                       //increase tree index to access next element 
                       #statIndexTreeArray += SINT_TO_UINT(#INCREMENT_BY_ONE);

                       //element was closed, pop index from stack
                       #statStackIndex -= SINT_TO_INT(#DECREMENT_BY_ONE);

                       //Set state, that should be executed after writing
                       #statFbNextState := #FB_STATE_CLOSE_STACK_ELEMENT;

                     ELSE
                       //close element with syntax key > as next element is child
                       // statInfoToWrite --> >
                       #statInfoToWrite := #XML_KEY_CLOSE_GREATER;
                       //Set state, that should be executed after writing
                       #statFbNextState := #FB_STATE_NEXT_ELEMENT;
                       //increase tree index to access next element 
                       #statIndexTreeArray += SINT_TO_UINT(#INCREMENT_BY_ONE);
                     END_IF;
                   END_IF;
                   //END Element
                 END_REGION ELEMENT

               ELSE // Undefined type provided
                 REGION UNDEFINED TYPE
                   #statStatus := #ERR_UNDEFINED_TYPE;
                 END_REGION UNDEFINED TYPE
             END_CASE;

             //Move to state Write
             #statFbState := #FB_STATE_WRITE_TO_XML;

           END_REGION WRITE VALUE

         #FB_STATE_CLOSE_STACK_ELEMENT: //Close Open Stack Elements
           REGION CLOSE ELEMENT FROM STACK
             //close element with syntax </key>

             IF #statStackIndex >= 0 THEN //more open elements available, not all elements are closed

               //statInfoToWrite --> </key>
               #statInfoToWrite := CONCAT(IN1 := #XML_KEY_OPEN,
                                          IN2 := #XML_KEY_CLOSE_SLASH,
                                          IN3 := #tree[#statStackIndexOpenElement[#statStackIndex]].key,
                                          IN4 := #XML_KEY_CLOSE_GREATER);

               //pop element from stack 
               #statStackIndex -= SINT_TO_INT(#DECREMENT_BY_ONE);

               IF #statStackIndex >= 0 THEN //more open elements available, not all elements are closed
                 //look at current stack item depth, if next tree element has 
                 IF NOT #statIsLastElement AND #tree[#statStackIndexOpenElement[#statStackIndex]].depth < #tree[#statIndexTreeArray + #NEXT_INDEX].depth THEN
                   //move to next element
                   #statFbNextState := #FB_STATE_NEXT_ELEMENT;
                   //increase tree index to access next element 
                   #statIndexTreeArray += SINT_TO_UINT(#INCREMENT_BY_ONE);
                 ELSE
                   //do nothing and return to fb state close element 
                   #statFbNextState := #FB_STATE_CLOSE_STACK_ELEMENT;
                 END_IF;

               ELSE
                 //no more open Elements, last Element was closed
                 #statIsLastElement := TRUE;

                 //only if this flag is set, can writer be finished
                 #statLastElementIsClosed := TRUE;

               END_IF;

             ELSE
               //no more open Elements, last Element was closed
               #statIsLastElement := TRUE;

               //only if this flag is set, can writer be finished
               #statLastElementIsClosed := TRUE;

             END_IF;
             //Move to state Write
             #statFbState := #FB_STATE_WRITE_TO_XML;
           END_REGION CLOSE ELEMENT FROM STACK

         #FB_STATE_WRITE_TO_XML: // Write to Byte Array
           REGION WRITE TO XML                
             //add information to xml byte array
             IF ((INT_TO_UINT(LEN(#statInfoToWrite)) + #statIndexXmlByteArray) < #statXmlByteLen) THEN
               Strg_TO_Chars(Strg := #statInfoToWrite,
                             pChars := #statIndexXmlByteArray,
                             Cnt => #tempCntCharsAdded,
                             Chars := #xmlByteArray);

               //move index of byte array 
               #statIndexXmlByteArray += #tempCntCharsAdded;
               //move to next state previously allocated
               #statFbState := #statFbNextState;
             ELSE // Error: Index out of bounds
               #statStatus := #ERR_XML_OUT_OF_BOUNDS;
             END_IF;

             IF #statLastElementIsClosed THEN
               //writer has written last information and execution is done
               #statStatus := #STATUS_EXECUTION_FINISHED;
               //current index equals count/size of xml byte array
               #statCount := #statIndexXmlByteArray;
             END_IF;
           END_REGION WRITE TO XML

         ELSE // Undefined state in state machine reached
           REGION UNDEFINED STATE
             #statStatus := #ERR_UNDEFINED_STATE;
           END_REGION UNDEFINED STATE                

       END_CASE;
       //Leave state machine if one of the following condition is true
       //1. state has not changed
       //2. error has occured
       //3. watchdog timer expired 
       //4. execution has finished
       // otherwise stay in state machine
     UNTIL (#statFbPreviousState = #statFbState OR #statStatus.%X15
       OR #instWatchdog.Q OR #statStatus = #STATUS_EXECUTION_FINISHED)
     END_REPEAT;
   END_REGION STATE_MACHINE

   REGION OUTPUTS
     // Write outputs
     IF (#statStatus = #STATUS_EXECUTION_FINISHED) AND (#statDone = FALSE) THEN // Execution finished without errors
       REGION EXECUTION FINSIHED
         #statDone := TRUE;
         #statBusy := FALSE;
         #statError := FALSE;
         // execution aborted --> set state no processing
         #statFbState := #FB_STATE_NO_PROCESSING;
       END_REGION EXECUTION FINSIHED

     ELSIF (#statStatus.%X15 = TRUE) AND (#statError = FALSE) THEN // Error occurred (#statStatus is 16#8000 to 16#FFFF)
       REGION ERROR OCCURED
         #statDone := FALSE;
         #statBusy := FALSE;
         #statError := TRUE;
         // execution aborted --> set state no processing
         #statFbState := #FB_STATE_NO_PROCESSING;
       END_REGION ERROR OCCURED

     ELSIF (#tempExecute = FALSE) AND ((#statDone = TRUE) OR (#statError = TRUE)) THEN // Reset outputs
       REGION EXECUTE RESETTED
         #statDone := FALSE;
         #statBusy := FALSE;
         #statError := FALSE;
         #statStatus := #STATUS_NO_CALL;
         // Reset application specific outputs
         #statCount := 0;
       END_REGION EXECUTE RESETTED
     END_IF;

     REGION WRITE STATIC VALUES TO OUTPUTS
       #done := #statDone;
       #busy := #statBusy;
       #error := #statError;
       #status := #statStatus;
       //  ENO mechanism is not used 
       ENO := TRUE;
       // Write application specific static values to outputs
       #count := #statCount;
     END_REGION WRITE STATIC VALUES TO OUTPUTS
   END_REGION OUTPUTS
END_FUNCTION_BLOCK

// folder: LStream/Utilities

FUNCTION "LStream_FindStringInByteCharArrayAdv" : DInt   // FC2, SCL
TITLE = LStream_FindStringInCharArrayAdv
{ S7_Optimized_Access := 'TRUE' }
AUTHOR : DI_FA_S_SUP_EuC
FAMILY : LStream
VERSION : 1.0
// Finds string in char array
   VAR_INPUT
      searchFor : String;   // Text that is searched for
      startPosition : DInt;   // Start position in array
   END_VAR
   VAR_IN_OUT
      searchIn : Array[*] of Byte;   // Array of Char to search in
   END_VAR
   VAR_TEMP
      tempLowerBound : DInt;   // Lower bound of given array
      tempNumElements : UDInt;   // Number of elements in given array
      tempLenSearchFor : Int;   // Length of text that is seached for
      tempPosInArray : DInt;   // Position in array during search (0-based)
      tempPosInString : Int;   // Position in working string during search
      tempString : String;   // Temporary string to work with
   END_VAR
   // Ret_Val : Returns the index of found string
   VAR CONSTANT
      FIRST_DIM : USInt := 1;   // Constant for first array dimenson
      MAX_LEN_STRING : UInt := 254;   // Max. length of String
   END_VAR
BEGIN
   REGION BLOCK INFO HEADER
     //===============================================================================
     // SIEMENS AG / (c)Copyright 2021
     //-------------------------------------------------------------------------------
     // Title:            LStream_FindStringInByteCharArrayAdv
     // Comment/Function: Searches for a specified string within an array of char
     // Library/Family:   LStream
     // Author:           DI FA S SUP E&C
     // Tested with:      S7-1500 V2.8
     // Engineering:      TIA Portal V16
     // Restrictions:     --
     // Requirements:     --
     //-------------------------------------------------------------------------------
     // Change log table:
     // Version  | Date       | Expert in charge | Changes applied
     //----------|------------|------------------|------------------------------------
     // 01.00.00 | 2021-03-10 |DI FA S SUP E&C   | First released version
     //===============================================================================
   END_REGION

   // Initialization
   #tempPosInString := 0;
   #tempPosInArray := #startPosition;
   #tempLenSearchFor := LEN(#searchFor);
   #LStream_FindStringInByteCharArrayAdv := -1;

   // Get number of elements
   #tempLowerBound := LOWER_BOUND(ARR := #searchIn, DIM := #FIRST_DIM);
   #tempNumElements := DINT_TO_UDINT(UPPER_BOUND(ARR := #searchIn, DIM := #FIRST_DIM) - #tempLowerBound + 1);

   IF (#tempPosInArray > #tempNumElements) THEN
       RETURN;
   END_IF;

   // Search for beginning of text until something was found and
   // as long as the index is less than the array size / number of elements in array
   WHILE ((#tempPosInString <= 0) AND (#tempPosInArray < #tempNumElements)) DO
       // Convert Chars to String
       Chars_TO_Strg(Chars := #searchIn,
                     pChars := #tempPosInArray,
                     Cnt := UDINT_TO_UINT(MIN(IN1 := #MAX_LEN_STRING, IN2 := #tempNumElements)),
                     Strg => #tempString);

       // Search for text at beginning
       #tempPosInString := FIND(IN1 := #tempString, IN2 := #searchFor);

       // Keyword was found
       IF #tempPosInString > 0 THEN
           // Output position of string
           #LStream_FindStringInByteCharArrayAdv := #tempLowerBound + #tempPosInArray + #tempPosInString - 1;
           EXIT;
       ELSE
           // Otherwise continue search in next string minus length of text at beginning to ensure
           // keywords are not broken up at the end of a string and thus missed
           #tempPosInArray += UINT_TO_INT(#MAX_LEN_STRING) - #tempLenSearchFor;
       END_IF;
   END_WHILE;
END_FUNCTION